// TIA Portal V18 export
FUNCTION_BLOCK "NoGoZoneV1"   // FB21, LAD
{ S7_Optimized_Access := 'TRUE' }
VERSION : 0.1
// stored: AutoNumber true, IsIECCheckEnabled false, IsRetainMemResEnabled false, MemoryReserve 100, SetENOAutomatically false, UDAEnableTagReadback false
   VAR_INPUT
      AutomateVersion : Int;
      MachineType : String;
      MachineLimit : Struct
         XSafety : Struct
            PosMax : DInt := 0;
            PosMin : DInt := 0;
            SafetyMargin : DInt;
            VelocityMax : DInt;
            VelocityMin : DInt;
         END_STRUCT;
         YSafety : Struct
            PosMax : DInt := 0;
            PosMin : DInt := 0;
            SafetyMargin : DInt;
            VelocityMax : DInt;
            VelocityMin : DInt;
         END_STRUCT;
         Z1Safety : Struct
            PosMax : DInt := 0;
            PosMin : DInt := 0;
            SafetyMargin : DInt;
            VelocityMax : DInt;
            VelocityMin : DInt;
         END_STRUCT;
         Z2Safety : Struct
            PosMax : DInt := 0;
            PosMin : DInt := 0;
            SafetyMargin : DInt;
            VelocityMax : DInt;
            VelocityMin : DInt;
         END_STRUCT;
         Heater : Struct
            FeedboxStart : DInt;
            FeedboxEnd : DInt;
            PrintboxStart : DInt;
            PrintboxEnd : DInt;
         END_STRUCT;
      END_STRUCT;
      XAxisHoming : Bool;
      YAxisHoming : Bool;
      Z1AxisHoming : Bool;
      Z2AxisHoming : Bool;
      ObjectHeight : DInt;   // Define object height
      ObjectWidth : DInt;   // Define object width
      ObjectMargin : DInt;   // Define object margin
      ObjectActivate : Bool;   // Use this to activate the No Go Zone
      XYstartendNormal : Struct
         XstartNormal : DInt;
         XendNormal : DInt;
         YstartNormal : DInt;
         YendNormal : DInt;
      END_STRUCT;
      XYstartendXL : Struct
         XstartXL : DInt;
         XendXL : DInt;
         YstartXL : DInt;
         YendXL : DInt;
      END_STRUCT;
      XActualPosition : DInt;
      YActualPosition : DInt;
      Z1ActualPosition : DInt;
      Z2ActualPosition : DInt;
   END_VAR
   VAR_OUTPUT
      NoGoAxisControl : Struct
         NoGoMotionLockXmove : Bool;
         NoGoMotionLockXjog : Bool;
         NoGoMotionLockYmove : Bool;
         NoGoMotionLockYjog : Bool;
         NoGoMotionLockZ1move : Bool;
         NoGoMotionLockZ1jog : Bool;
         NoGoMotionLockZ2move : Bool;
         NoGoMotionLockZ2jog : Bool;
         NoGoHomingPermissionX : Bool;
         NoGoHomingPermissionY : Bool;
         NoGoHomingPermissionZ1 : Bool;
         NoGoHomingPermissionZ2 : Bool;
         NoGoAlwaysMove : Bool;
      END_STRUCT;
      NoGoStatus : Struct
         NoGoZoneActive : Bool;
         YouAreInNoGoZoneWarning : Bool;
         NoGoZoneCollisionError : Bool;
      END_STRUCT;
   END_VAR
   VAR
      internalNoGoZoneXY : Struct
         internalNoGoZoneXstart : DInt;
         internalNoGoZoneXend : DInt;
         internalNoGoZoneYstart : DInt;
         internalNoGoZoneYend : DInt;
      END_STRUCT;
      internalNoGoZoneZ1start : DInt;
      internalNoGoZoneZ1end : DInt;
      internalNoGoZoneZ2start : DInt;
      internalNoGoZoneZ2end : DInt;
      internalObjectWithMargin : DInt;
      ControlCondition01 : Bool;   // Checking if condition 1 is fine
      ControlCondition02 : Bool;   // Checking if condition 2 is fine
      ControlCondition03 : Bool;   // Checking if condition 3 is fine
   END_VAR
BEGIN

REGION Network 1: Zone Active
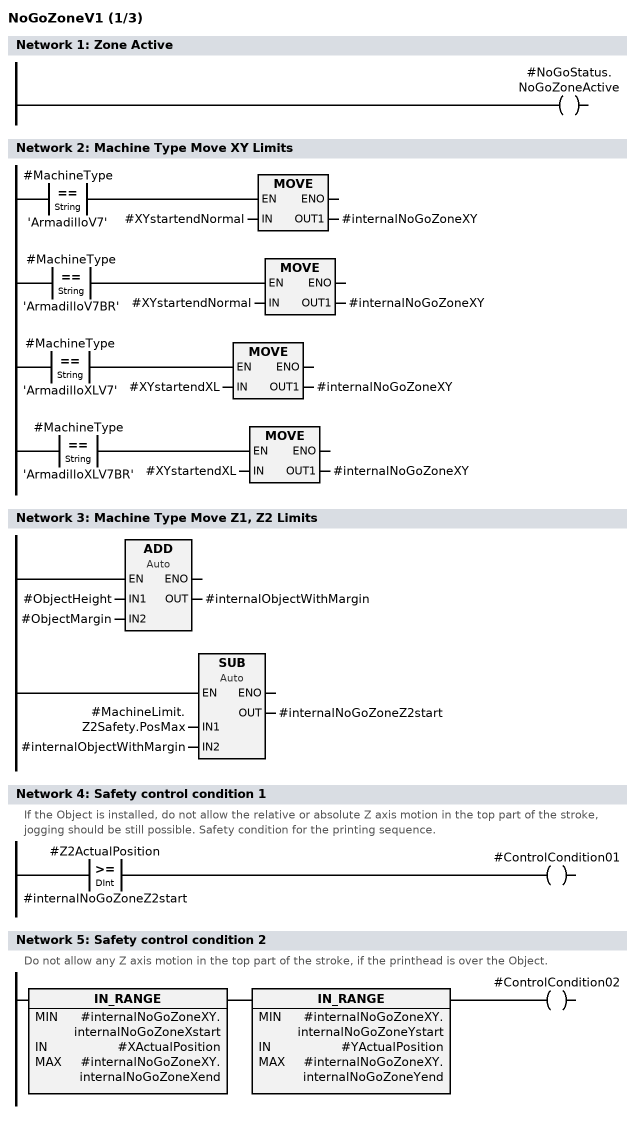
   RUNG wire#powerrail
      Coil( #NoGoStatus.NoGoZoneActive )
   END_RUNG
   // the same network as SCL:
   #NoGoStatus.NoGoZoneActive := TRUE;
END_REGION

REGION Network 2: Machine Type Move XY Limits
   RUNG wire#powerrail
      { S7_Templates := "SrcType := String" } EQ_Contact(in1 := #MachineType, in2 := 'ArmadilloV7')
      Move(in := #XYstartendNormal, out1 => #internalNoGoZoneXY)
   END_RUNG
   RUNG wire#powerrail
      { S7_Templates := "SrcType := String" } EQ_Contact(in1 := #MachineType, in2 := 'ArmadilloV7BR')
      Move(in := #XYstartendNormal, out1 => #internalNoGoZoneXY)
   END_RUNG
   RUNG wire#powerrail
      { S7_Templates := "SrcType := String" } EQ_Contact(in1 := #MachineType, in2 := 'ArmadilloXLV7')
      Move(in := #XYstartendXL, out1 => #internalNoGoZoneXY)
   END_RUNG
   RUNG wire#powerrail
      { S7_Templates := "SrcType := String" } EQ_Contact(in1 := #MachineType, in2 := 'ArmadilloXLV7BR')
      Move(in := #XYstartendXL, out1 => #internalNoGoZoneXY)
   END_RUNG
   // the same network as SCL:
   IF #MachineType = 'ArmadilloV7' THEN #internalNoGoZoneXY := #XYstartendNormal; END_IF;
   IF #MachineType = 'ArmadilloV7BR' THEN #internalNoGoZoneXY := #XYstartendNormal; END_IF;
   IF #MachineType = 'ArmadilloXLV7' THEN #internalNoGoZoneXY := #XYstartendXL; END_IF;
   IF #MachineType = 'ArmadilloXLV7BR' THEN #internalNoGoZoneXY := #XYstartendXL; END_IF;
END_REGION

REGION Network 3: Machine Type Move Z1, Z2 Limits
   RUNG wire#powerrail
      Add(in1 := #ObjectHeight, in2 := #ObjectMargin, out => #internalObjectWithMargin)
   END_RUNG
   RUNG wire#powerrail
      Sub(in1 := #MachineLimit.Z2Safety.PosMax, in2 := #internalObjectWithMargin, out => #internalNoGoZoneZ2start)
   END_RUNG
   // the same network as SCL:
   #internalObjectWithMargin := #ObjectHeight + #ObjectMargin;
   #internalNoGoZoneZ2start := #MachineLimit.Z2Safety.PosMax - #internalObjectWithMargin;
END_REGION

REGION Network 4: Safety control condition 1
   // If the Object is installed, do not allow the relative or absolute Z axis motion in the top part of the stroke, jogging should be still possible. Safety condition for the printing sequence.
   RUNG wire#powerrail
      { S7_Templates := "SrcType := DInt" } GE_Contact(in1 := #Z2ActualPosition, in2 := #internalNoGoZoneZ2start)
      Coil( #ControlCondition01 )
   END_RUNG
   // the same network as SCL:
   #ControlCondition01 := #Z2ActualPosition >= #internalNoGoZoneZ2start;
END_REGION

REGION Network 5: Safety control condition 2
   // Do not allow any Z axis motion in the top part of the stroke, if the printhead is over the Object.
   RUNG wire#powerrail
      { S7_Templates := "SrcType := DInt" } InRange(min := #internalNoGoZoneXY.internalNoGoZoneXstart, in := #XActualPosition, max := #internalNoGoZoneXY.internalNoGoZoneXend)
      { S7_Templates := "SrcType := DInt" } InRange(min := #internalNoGoZoneXY.internalNoGoZoneYstart, in := #YActualPosition, max := #internalNoGoZoneXY.internalNoGoZoneYend)
      Coil( #ControlCondition02 )
   END_RUNG
   // the same network as SCL:
   #ControlCondition02 := (#internalNoGoZoneXY.internalNoGoZoneXstart <= #XActualPosition) AND (#XActualPosition <= #internalNoGoZoneXY.internalNoGoZoneXend) AND (#internalNoGoZoneXY.internalNoGoZoneYstart <= #YActualPosition) AND (#YActualPosition <= #internalNoGoZoneXY.internalNoGoZoneYend);
END_REGION

REGION Network 6: Safety control condition 3
   // Do not allow any motion when the Object is in a collision with axes.
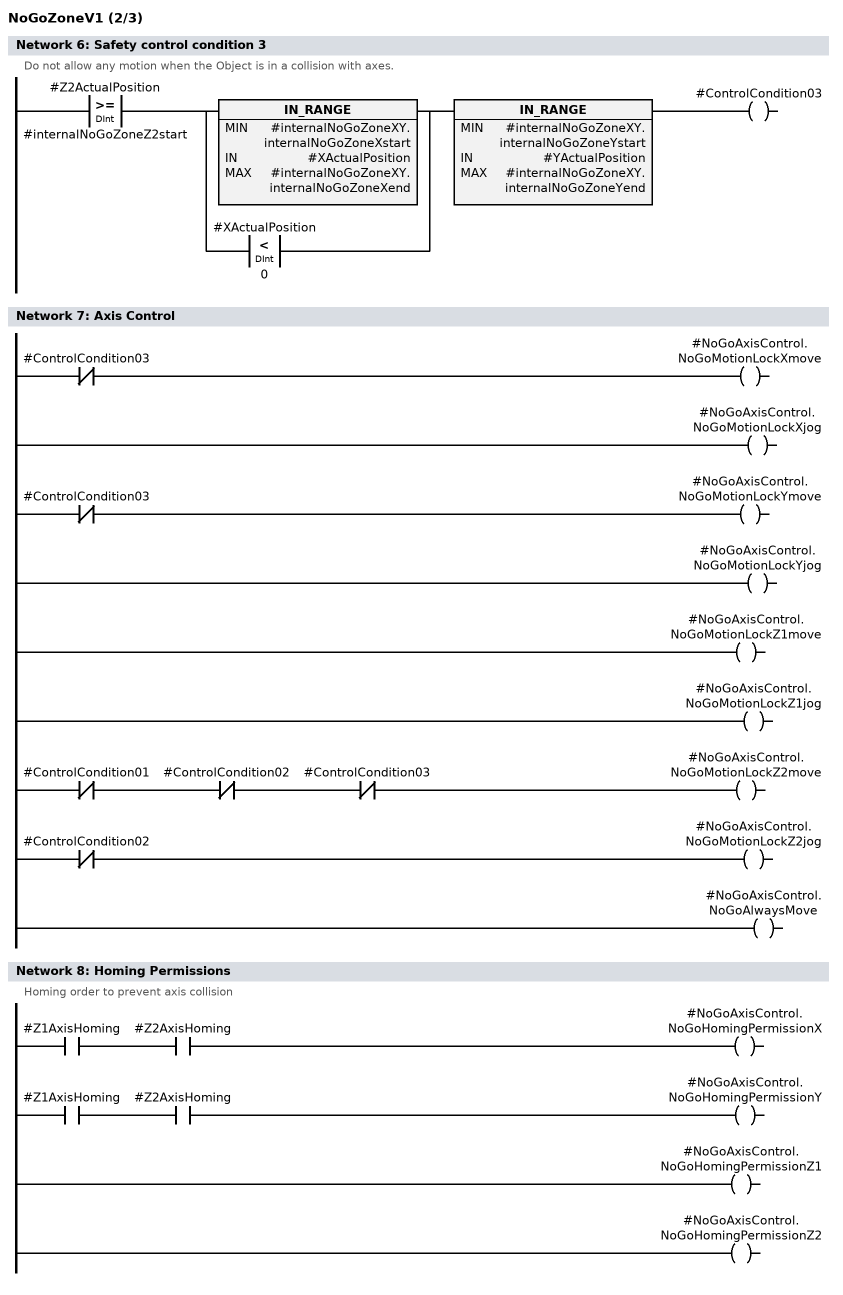
   RUNG wire#powerrail
      { S7_Templates := "SrcType := DInt" } GE_Contact(in1 := #Z2ActualPosition, in2 := #internalNoGoZoneZ2start)
      wire#w1
      { S7_Templates := "SrcType := DInt" } InRange(min := #internalNoGoZoneXY.internalNoGoZoneXstart, in := #XActualPosition, max := #internalNoGoZoneXY.internalNoGoZoneXend)
      wire#w2
      { S7_Templates := "SrcType := DInt" } InRange(min := #internalNoGoZoneXY.internalNoGoZoneYstart, in := #YActualPosition, max := #internalNoGoZoneXY.internalNoGoZoneYend)
      Coil( #ControlCondition03 )
   END_RUNG
   RUNG wire#w1
      { S7_Templates := "SrcType := DInt" } LT_Contact(in1 := #XActualPosition, in2 := 0)
   END_RUNG wire#w2
   // the same network as SCL:
   #ControlCondition03 := (#Z2ActualPosition >= #internalNoGoZoneZ2start) AND (((#internalNoGoZoneXY.internalNoGoZoneXstart <= #XActualPosition) AND (#XActualPosition <= #internalNoGoZoneXY.internalNoGoZoneXend)) OR (#XActualPosition < 0)) AND (#internalNoGoZoneXY.internalNoGoZoneYstart <= #YActualPosition) AND (#YActualPosition <= #internalNoGoZoneXY.internalNoGoZoneYend);
END_REGION

REGION Network 7: Axis Control
   RUNG wire#powerrail
      I_Contact( #ControlCondition03 )
      Coil( #NoGoAxisControl.NoGoMotionLockXmove )
   END_RUNG
   RUNG wire#powerrail
      Coil( #NoGoAxisControl.NoGoMotionLockXjog )
   END_RUNG
   RUNG wire#powerrail
      I_Contact( #ControlCondition03 )
      Coil( #NoGoAxisControl.NoGoMotionLockYmove )
   END_RUNG
   RUNG wire#powerrail
      Coil( #NoGoAxisControl.NoGoMotionLockYjog )
   END_RUNG
   RUNG wire#powerrail
      Coil( #NoGoAxisControl.NoGoMotionLockZ1move )
   END_RUNG
   RUNG wire#powerrail
      Coil( #NoGoAxisControl.NoGoMotionLockZ1jog )
   END_RUNG
   RUNG wire#powerrail
      I_Contact( #ControlCondition01 )
      I_Contact( #ControlCondition02 )
      I_Contact( #ControlCondition03 )
      Coil( #NoGoAxisControl.NoGoMotionLockZ2move )
   END_RUNG
   RUNG wire#powerrail
      I_Contact( #ControlCondition02 )
      Coil( #NoGoAxisControl.NoGoMotionLockZ2jog )
   END_RUNG
   RUNG wire#powerrail
      Coil( #NoGoAxisControl.NoGoAlwaysMove )
   END_RUNG
   // the same network as SCL:
   #NoGoAxisControl.NoGoMotionLockXmove := NOT #ControlCondition03;
   #NoGoAxisControl.NoGoMotionLockXjog := TRUE;
   #NoGoAxisControl.NoGoMotionLockYmove := NOT #ControlCondition03;
   #NoGoAxisControl.NoGoMotionLockYjog := TRUE;
   #NoGoAxisControl.NoGoMotionLockZ1move := TRUE;
   #NoGoAxisControl.NoGoMotionLockZ1jog := TRUE;
   #NoGoAxisControl.NoGoMotionLockZ2move := NOT #ControlCondition01 AND NOT #ControlCondition02 AND NOT #ControlCondition03;
   #NoGoAxisControl.NoGoMotionLockZ2jog := NOT #ControlCondition02;
   #NoGoAxisControl.NoGoAlwaysMove := TRUE;
END_REGION

REGION Network 8: Homing Permissions
   // Homing order to prevent axis collision
   RUNG wire#powerrail
      Contact( #Z1AxisHoming )
      Contact( #Z2AxisHoming )
      Coil( #NoGoAxisControl.NoGoHomingPermissionX )
   END_RUNG
   RUNG wire#powerrail
      Contact( #Z1AxisHoming )
      Contact( #Z2AxisHoming )
      Coil( #NoGoAxisControl.NoGoHomingPermissionY )
   END_RUNG
   RUNG wire#powerrail
      Coil( #NoGoAxisControl.NoGoHomingPermissionZ1 )
   END_RUNG
   RUNG wire#powerrail
      Coil( #NoGoAxisControl.NoGoHomingPermissionZ2 )
   END_RUNG
   // the same network as SCL:
   #NoGoAxisControl.NoGoHomingPermissionX := #Z1AxisHoming AND #Z2AxisHoming;
   #NoGoAxisControl.NoGoHomingPermissionY := #Z1AxisHoming AND #Z2AxisHoming;
   #NoGoAxisControl.NoGoHomingPermissionZ1 := TRUE;
   #NoGoAxisControl.NoGoHomingPermissionZ2 := TRUE;
END_REGION

REGION Network 9: Status
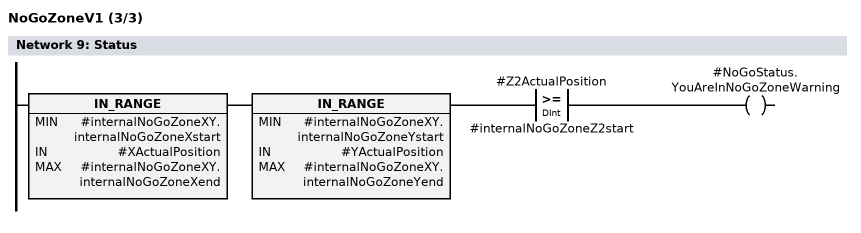
   RUNG wire#powerrail
      { S7_Templates := "SrcType := DInt" } InRange(min := #internalNoGoZoneXY.internalNoGoZoneXstart, in := #XActualPosition, max := #internalNoGoZoneXY.internalNoGoZoneXend)
      { S7_Templates := "SrcType := DInt" } InRange(min := #internalNoGoZoneXY.internalNoGoZoneYstart, in := #YActualPosition, max := #internalNoGoZoneXY.internalNoGoZoneYend)
      { S7_Templates := "SrcType := DInt" } GE_Contact(in1 := #Z2ActualPosition, in2 := #internalNoGoZoneZ2start)
      Coil( #NoGoStatus.YouAreInNoGoZoneWarning )
   END_RUNG
   // the same network as SCL:
   #NoGoStatus.YouAreInNoGoZoneWarning := (#internalNoGoZoneXY.internalNoGoZoneXstart <= #XActualPosition) AND (#XActualPosition <= #internalNoGoZoneXY.internalNoGoZoneXend) AND (#internalNoGoZoneXY.internalNoGoZoneYstart <= #YActualPosition) AND (#YActualPosition <= #internalNoGoZoneXY.internalNoGoZoneYend) AND (#Z2ActualPosition >= #internalNoGoZoneZ2start);
END_REGION
END_FUNCTION_BLOCK
